// Acknowledge all event class related objects.
FUNCTION F_AcknowledgeEventClass  
VAR_INPUT
	nEventClassID		: UINT					:= 0;		// Target event class ID.
END_VAR
VAR
	_iObj				: I_BA_Object;
	_iEvtObj			: I_BA_EventObject;
END_VAR

// Iterate over all objects:
WHILE (F_BA_IterateObjects(_iObj)) DO
	IF (NOT __QUERYINTERFACE(_iObj,_iEvtObj)) THEN
		;	     
	ELSIF (_iEvtObj.EventClassID <> nEventClassID) THEN
		; // Skip.
	ELSE
		_iEvtObj.AcknowledgeRm := TRUE;
	END_IF
END_WHILE

END_FUNCTION

(* stored: Version 1.1.0.1, ProductVersion 3.1.4024.12
   POU F_AcknowledgeEventClass: Id {89fd74b8-e45b-4b4a-8f6d-88c66b5fc523}, SpecialFunc None *)
